_CFC_ (* Continuous Function Chart, elements in execution order *)
#0 SUB(SCHU_P2_4_M_MAXSPEED_PE, SCHU_P2_4_SPEEDMOTOR)
#1 ABS(#0)
#2 >(#1, 0.3)
#3 AND(SCHU_P2_4_PE_PID_VKL, #2)
#4 <>(SCHU_P2_4_M_MAXSPEED_CH, SCHU_P2_4_M_MAXSPEED_CH_OLD)
#5 AND(#4, NOT SCHU_P2_4_PE_PID_VKL)
#6 OR(#3, #5)
#7 RS_RUCH:RS(SET: #6, RESET1: #9.Q)
#8 V_RUCH <= #7.Q1
#9 TON_RUCH:TON(IN: #7.Q1, PT: T#10s)
#10 <>(SCHU_P2_4_M_MAXSPEED_PE, 0)
#11 AND(SCHU_P2_4_PE_PID_VKL, #10)
#12 Zad_PE:TON(IN: #11, PT: T#2s)
#13 SEL(#12.Q, SCHU_P2_4_M_MAXSPEED_CH, SCHU_P2_4_M_MAXSPEED_PE)
#14 SCHU_P2_4_M_MAXSPEED <= #13
#15 AND(SCHU_P2_4_YA2_M_UST_VKL_UVEL_CHAST, SCHU_P2_4_YA3_M_UST_VKL_UVEL_CHAST, SCHU_P2_4_YA4_M_UST_VKL_UVEL_CHAST, SCHU_P2_4_UST_RE_RABOTA)
#16 TON_STER_1:TON(IN: #15, PT: T#60s)
#17 OR(#16.Q, SCHU_P2_4_M_SB2_STER_REG)
#18 AND(#17, SCHU_P2_4_UST_RE_RABOTA, NOT V_RUCH)
#19 OR(V_RUCH, SCHU_P2_4_UST_RE_PUSK)
#20 SEL(#18, SCHU_P2_4_SPEEDMOTOR, SCHU_P2_4_M_MAXSPEED)
#21 AND(NOT SCHU_P2_4_SA8_DI4_M, SCHU_P2_4_SA1_DI6_M)
#22 AND(#18, NOT V_RUCH)
#23 SEL(#22, SCHU_P2_4_M_USKORENIE_PUSK, SCHU_P2_4_M_USKORENIE_UPR)
#24 OR(SCHU_P2_4_YA2_B_UST_VKL_STER_REG, SCHU_P2_4_YA3_B_UST_VKL_STER_REG, SCHU_P2_4_YA4_B_UST_VKL_STER_REG)
#25 AND(SCHU_P2_4_UST_RE_RABOTA, #24)
#26 TON_STER_2:TON(IN: #25, PT: T#60s)
#27 AND(NOT SCHU_P2_4_M_SB2_STER_REG, #26.Q, SCHU_P2_4_UST_RE_RABOTA, NOT V_RUCH)
#28 SEL(#27, #20, SCHU_P2_4_M_MINSPEED)
#29 SEL(#19, #28, SCHU_P2_4_M_MAXSPEED)
#30 SEL(SCHU_P2_4_UST_SOST_VKL, 0, #29)
#31 AND(SCHU_P2_4_SA8_DI4_M, NOT SCHU_P2_4_SA1_DI6_M)
#32 AND(#27, NOT V_RUCH)
#33 SEL(#32, SCHU_P2_4_M_ZAMEDLENIE_OST, SCHU_P2_4_M_ZAMEDLENIE_UPR)
#34 SEL(SCHU_P2_4_UST_SET_STOP, #33, 1000)
#35 RR:RAMP_REAL(#30, #23, #34, T#1s, -)
#36 SCHU_P2_4_SPEEDMOTOR <= #35
#37 MOVE(EN: SCHU_P2_4_SA1_DO1, #35)
#38 SEL(#37.ENO, 0, #37)
#39 SEL(#21, #38, SCHU_P2_4_M_ZAD_RUCH)
#40 SCHU_P2_4_M1_ZAD_VN <= #39
#41 MOVE(EN: SCHU_P2_4_SA8_DO8, #35)
#42 SEL(#41.ENO, 0, #41)
#43 SEL(#31, #42, SCHU_P2_4_M_ZAD_RUCH)
#44 SCHU_P2_4_M2_ZAD_VN <= #43
#45 SCHU_P2_4_PE1_UST_OLD <= SCHU_P2_4_PE1_UST
#46 SCHU_P2_4_M_MAXSPEED_CH_OLD <= SCHU_P2_4_M_MAXSPEED_CH
#47 RT_KOMVKL_2:R_TRIG(CLK: TRUE)
#48 MOVE(EN: #47.Q, 5)
#49 SCHU_P2_4_M_ZAD_RUCH <= #48
_END_CFC_
END_PROGRAM

(* POU IM/P1_Upr, CFC *)
PROGRAM P1_Upr
VAR
	fb_HVACMS_P1: FB_HVACMotor1Speed;
	SR_P1: SR;
	startDelay_P1: TIME := T#0s;
	stopDelay_P1: TIME := T#0s;
	delayFBC_P1: TIME;
	feedbPT_P1: TIME :=T#10s ;
	delayFBP_P1: TIME := T#10s;
	TON_P1_OTKL_Leto: TON;
	TON_P1_VKL_Leto: TON;
END_VAR
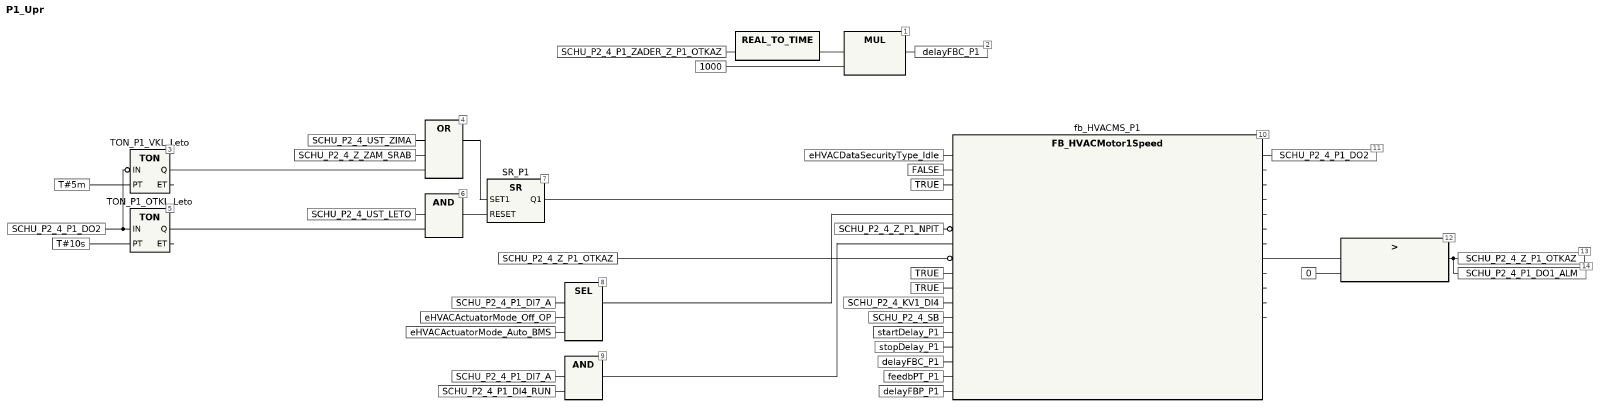
_CFC_ (* Continuous Function Chart, elements in execution order *)
#0 REAL_TO_TIME(SCHU_P2_4_P1_ZADER_Z_P1_OTKAZ)
#1 MUL(#0, 1000)
#2 delayFBC_P1 <= #1
#3 TON_P1_VKL_Leto:TON(IN: NOT SCHU_P2_4_P1_DO2, PT: T#5m)
#4 OR(SCHU_P2_4_UST_ZIMA, SCHU_P2_4_Z_ZAM_SRAB, #3.Q)
#5 TON_P1_OTKL_Leto:TON(IN: SCHU_P2_4_P1_DO2, PT: T#10s)
#6 AND(SCHU_P2_4_UST_LETO, #5.Q)
#7 SR_P1:SR(SET1: #4, RESET: #6)
#8 SEL(SCHU_P2_4_P1_DI7_A, eHVACActuatorMode_Off_OP, eHVACActuatorMode_Auto_BMS)
#9 AND(SCHU_P2_4_P1_DI7_A, SCHU_P2_4_P1_DI4_RUN)
#10 fb_HVACMS_P1:FB_HVACMotor1Speed(eHVACDataSecurityType_Idle, FALSE, TRUE, #7.Q1, #8, NOT SCHU_P2_4_Z_P1_NPIT, #9, NOT SCHU_P2_4_Z_P1_OTKAZ, TRUE, TRUE, SCHU_P2_4_KV1_DI4, SCHU_P2_4_SB, startDelay_P1, stopDelay_P1, delayFBC_P1, feedbPT_P1, delayFBP_P1)
#11 SCHU_P2_4_P1_DO2 <= #10.out 1
#12 >(#10.out 8, 0)
#13 SCHU_P2_4_Z_P1_OTKAZ <= #12
#14 SCHU_P2_4_P1_DO1_ALM <= #12
_END_CFC_
END_PROGRAM

(* POU IM/P2_Upr, CFC *)
PROGRAM P2_Upr
VAR
	fb_HVACMS_P2: FB_HVACMotor1Speed;
	startDelay_P2: TIME := T#0s;
	stopDelay_P2: TIME := T#0s;
	delayFBC_P2: TIME := T#10s;
	feedbPT_P2: TIME :=T#10s ;
	delayFBP_P2: TIME := T#10s;
	errorGeneral: BOOL;
	RS_UE2_SHU1_P1_2_P2_DO3: RS;
	RS_UE3_SHU1_P1_2_P2_DO3: RS;
	UE3_VLmYST: BOOL;
END_VAR
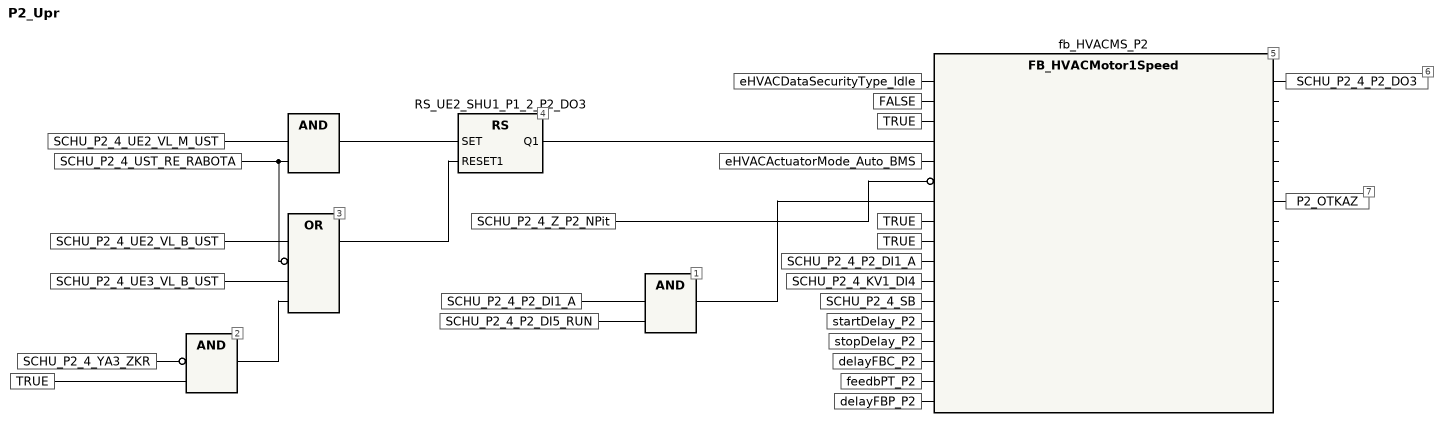
_CFC_ (* Continuous Function Chart, elements in execution order *)
#0 AND(SCHU_P2_4_UE2_VL_M_UST, SCHU_P2_4_UST_RE_RABOTA)
#1 AND(SCHU_P2_4_P2_DI1_A, SCHU_P2_4_P2_DI5_RUN)
#2 AND(NOT SCHU_P2_4_YA3_ZKR, TRUE)
#3 OR(SCHU_P2_4_UE2_VL_B_UST, NOT SCHU_P2_4_UST_RE_RABOTA, SCHU_P2_4_UE3_VL_B_UST, #2)
#4 RS_UE2_SHU1_P1_2_P2_DO3:RS(SET: #0, RESET1: #3)
#5 fb_HVACMS_P2:FB_HVACMotor1Speed(eHVACDataSecurityType_Idle, FALSE, TRUE, #4.Q1, eHVACActuatorMode_Auto_BMS, NOT SCHU_P2_4_Z_P2_NPit, #1, TRUE, TRUE, SCHU_P2_4_P2_DI1_A, SCHU_P2_4_KV1_DI4, SCHU_P2_4_SB, startDelay_P2, stopDelay_P2, delayFBC_P2, feedbPT_P2, delayFBP_P2)
#6 SCHU_P2_4_P2_DO3 <= #5.out 1
#7 P2_OTKAZ <= #5.out 7
_END_CFC_
END_PROGRAM

(* POU IM/YA1_Upr, CFC *)
PROGRAM YA1_Upr
VAR
	RS_YA1_Open: RS;
	RT_Pusk: R_TRIG;
	RT_OSTANOV: R_TRIG;
	fb_HVACPA: FB_HVAC2PointActuator;

	stokeTime: TIME;
	enableLimitSwitch: BOOL := TRUE;
	FT_PCH_OTKL: R_TRIG;
	TON_PCH_OTKL: TON;
	ZADERJ_SHOD_YA1: TON;
	TON_YA1_Z_ZAM_TE2: TON;
	TON_OTK_MV: TON;
END_VAR
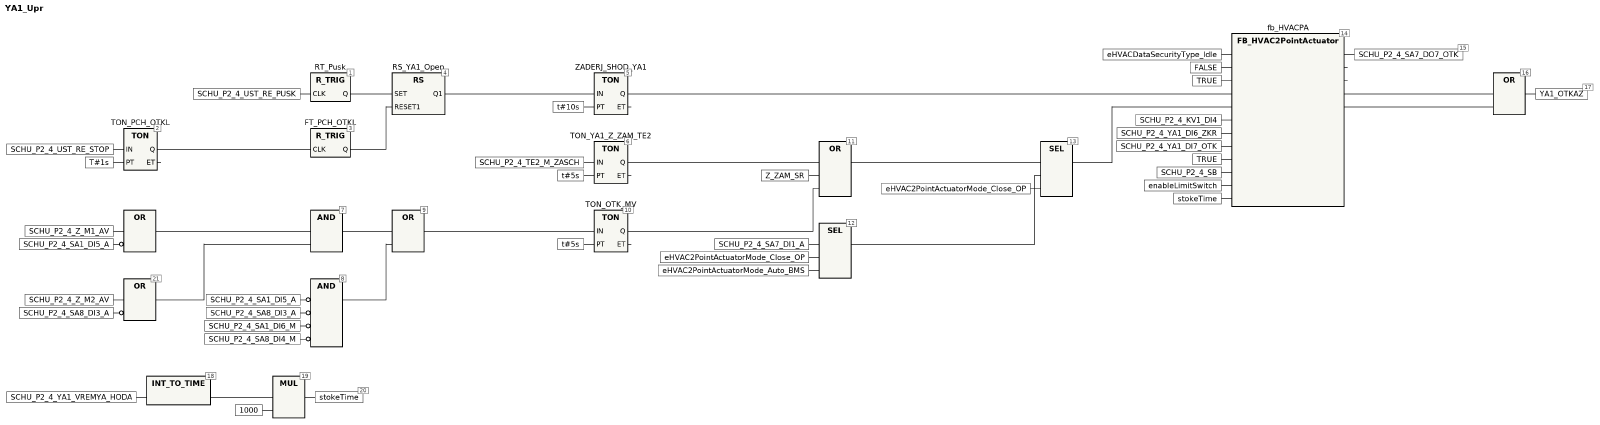
